PROGRAM MAIN
VAR
END_VAR

END_PROGRAM

(* stored: Version 1.1.0.1
   POU MAIN: Id {6fbd2007-8739-46f0-8ac3-c75236c8751b} *)
